// TwinCAT 3 PLC project PLC1
// ProgramVersion: 3.1.4026.19
// libraries:
//   Tc2_MC2, * (Beckhoff Automation GmbH)
//   Tc2_Standard, * (Beckhoff Automation GmbH)
//   Tc2_System, * (Beckhoff Automation GmbH)
// project tree:
//   GVLs/ Analog_Variables.TcGVL, Global_Variables.TcGVL, GVL_Axes.TcGVL
//   / PlcTask.TcTTO
//   POUs/ Analog_PRG.TcPOU, MAIN.TcPOU, Servo_Details.TcPOU, Step_3_Unscrambler.TcPOU, Step_4_EvenEnder.TcPOU, Step_5_Grading.TcPOU, Step_6_Log_Sequence.TcPOU, Step_7_Saw_Positioning.TcPOU, Step_8_Outfeed.TcPOU, Tower_Light_Manager.TcPOU, Step_1_TiltHoist.TcPOU, Step_2_StickMachine.TcPOU
// real-time tasks:
//   TASK PlcTask: cycle T#10ms, priority 20, ADS port 350
// motion (NC):
//   TASK NC-Task 1 SAF: cycle T#2ms, priority 4, ADS port 501
//   TASK NC-Task 1 SVB: cycle T#10ms, priority 8, ADS port 511
//   AXIS Axis 1 (id 1)
//     Dynamic: Acceleration=4141.08, Deceleration=4141.08, Jerk=45551.9
//     Velo: RefSearch=37.6461354666667, RefSync=37.6461354666667, SlowManual=188.230677333333, FastManual=1129.384064, Fast=3764.61354666667, Maximum=3764.61
//     PositionAreaControl: Enable=false
//     TargetPosControl: Range=0.5, Time=0.01
//     OtherSettings: AllowMotionCmdToSlave=true
//     encoder EncType=8
//       EncPara: ScaleFactorNumerator=104.8576, ScaleFactorDenominator=1048576, MaxCount=#xffffffff
//     drive DrvType=9
//       DrvPara: MaxCount=#xffffffff, DriveControlDWord=#x00030000
//         Analog: VeloReferenz=4141.07490133333, VeloScale=1.02398817080127, TorqueSetpointScale=10, ScaleFactorActTorque=0.1
//         TimeComp: TaskDelayCycles=1
//     controller CtrType=1
//       CtrPara: PriorControlFactor=1
//         PosDiffControl: Enable=false
//         PID: PosKp=10
//         Observer: BandWidth=20
// I/O:
//   DEVICE Device 1 (EtherCAT), AmsNetId 5.164.185.153.2.1
//     Term 1 (EK1100) [EK1100 EtherCAT Coupler (2A E-Bus)]
//       Term 2 (EL1417) [EL1417 32Ch. Dig. Input 24V]
//       Term 3 (EL2407) [EL2407 32Ch. Dig. Output 24V, 0.5A]
//       Term 9 (EL9011) [EL9011 End Terminal]
//     Drive 4 (AX5203-0000-0011) [AX5203-0000-0011 EtherCAT Drive (SoE, 2 Ch.)]
// variable links:
//   NC-Task 1 SAF/Axes/Axis 1 <-> Device 1 (EtherCAT)/Drive 4 (AX5203-0000-0011)
//     Drive/Inputs/In/nDcOutputTime <-> InfoData/DcOutputShift
//     Drive/Inputs/In/nState1 <-> AT 1/Drive status word @bit 8
//     Drive/Inputs/In/nState2 <-> AT 1/Drive status word
//     Drive/Inputs/In/nState4 @bit 1 <-> WcState/InputToggle
//     Drive/Inputs/In/nState4 <-> WcState/WcState
//     Drive/Outputs/Out/nCtrl1 <-> MDT 1/Master control word @bit 8
//     Drive/Outputs/Out/nDataOut2 <-> MDT 1/Velocity command value
//     Enc/Inputs/In/nDataIn1 <-> AT 1/Position feedback 1 value
//     Enc/Inputs/In/nDcInputTime <-> InfoData/DcInputShift
//     Enc/Inputs/In/nState4 @bit 1 <-> WcState/InputToggle
//     Enc/Inputs/In/nState4 <-> WcState/WcState
//   PLC1/PLC1 Instance <-> NC-Task 1 SAF/Axes/Axis 1
//     PlcTask Inputs/GVL_Axes.Axis1.NcToPlc <-> Outputs/ToPlc
//     PlcTask Outputs/GVL_Axes.Axis1.PlcToNc <-> Inputs/FromPlc

CONFIGURATION PLC1
    RESOURCE PLC ON TwinCAT3
        TASK PlcTask(INTERVAL := T#10ms, PRIORITY := 20);
        PROGRAM MAIN WITH PlcTask : MAIN;
        PROGRAM Step_1_TiltHoist WITH PlcTask : Step_1_TiltHoist;
        PROGRAM Step_2_StickMachine WITH PlcTask : Step_2_StickMachine;
        PROGRAM Step_3_Unscrambler WITH PlcTask : Step_3_Unscrambler;
        PROGRAM Step_4_EvenEnder WITH PlcTask : Step_4_EvenEnder;
        PROGRAM Servo_Details WITH PlcTask : Servo_Details;
        PROGRAM Step_5_Grading WITH PlcTask : Step_5_Grading;
        PROGRAM Step_6_Log_Sequence WITH PlcTask : Step_6_Log_Sequence;
        PROGRAM Step_7_Saw_Positioning WITH PlcTask : Step_7_Saw_Positioning;
        PROGRAM Step_8_Outfeed WITH PlcTask : Step_8_Outfeed;
    END_RESOURCE
END_CONFIGURATION

// ---- GVLs/Analog_Variables.TcGVL
VAR_GLOBAL
	

	AI_INT  : INT;   // from EL3255, 0.0–10.0 V
    AO_INT : INT;   // to EL4004, 0.0–10.0 V



















END_VAR

// ---- GVLs/Global_Variables.TcGVL
VAR_GLOBAL 
//--------------------------------- Power_Panel_IO---------------------------------


	//INPUTS for EL1409 (16 inputs avilable)
	SawPhotoeye AT %I*:BOOL;
	OutfeedRopePull AT %I*:BOOL;
	//Manual Motor Protector Signals//
	TiltHoistMMP AT %I*:BOOL;
	StickConveyorMMP AT %I*:BOOL; 
	StickFeedChainMMP AT %I*:BOOL; 
	EvenEnderMMP AT %I*:BOOL; 
	ScrapConveyorMMP AT %I*:BOOL; 
	OutFeedConveyorMMP AT %I*:BOOL;
	DustCollectorMMP AT %I*:BOOL;
	SawBlade1MMP AT %I*:BOOL;
	SawBlade2MMP AT %I*:BOOL;
	//Safety Singal
	SafetyCircuitSignal AT %I*:BOOL;
	
		//Servo
		OverTRavelLimitREV AT %I*:BOOL; 
		OverTRavelLimitFWD AT %I*:BOOL;
		HomingSensor AT %I*:BOOL;
	

	//INPUTS for EL1859 (8 inputs avilable)
	VFD1Faulted AT %I*:BOOL; //Unscrambler Chain
	VFD2Faulted AT %I*:BOOL; //Grading Chain 
	VFD3Faulted AT %I*:BOOL; //Feed Chain - Saw
	GradingEndLimit AT %I*:BOOL; // Grading end limit switch
	SawFeedChainHomingSensor AT %I*:BOOL; // saw feed chain homing sensor	
	
	//OUTPUTS for EL2409 (16 outputs avilable)
	ResetVFDs AT %Q*:BOOL;
	UnscramblerVFD1FWD AT %Q*:BOOL; //Unscrambler Chain FWD
	UnscramblerVFD1REV AT %Q*:BOOL; //Unscrambler Chain REV
	GradingVFD2FWD AT %Q*:BOOL; //Grading Chain 
	SawFeedChainVFD3FWD AT %Q*:BOOL; //Feed Chain - Saw
	
	TiltHoistFWD AT %Q*:BOOL;
	TiltHoistREV AT %Q*:BOOL;
	StickConveyorFWD AT %Q*:BOOL;
	StickFeedChainFWD AT %Q*:BOOL;
	EvenEnderFWD AT %Q*:BOOL;
	ScrapConveyorFWD AT %Q*:BOOL;
	OutFeedConveyorFWD AT %Q*:BOOL;
	DustCollectorFWD AT %Q*:BOOL;
	SawBladesFWD AT %Q*:BOOL;
	
	//OUTPUTS for EL1859 (8 outputs available)
	GradingVFD2REV AT %Q*:BOOL; //Grading Chain REV
	SawFeedChainVFD3REV AT %Q*:BOOL; //Feed Chain - Saw
	
	
	
//---------------------------------Control_Panel_IO----------------------------------

	
	//INPUTS for EL1409
	
	PBFoot:ARRAY[4..16] OF BOOL;
	
	ConfirmPB AT %I*:BOOL; //Confirms Board Input
	CancelPB AT %I*:BOOL; //Cancels Last Board Input
	//PanelStopPB AT %I*:BOOL; //CycleStopPB same input 
	
	//OUTPUTS for EL2409

	
	LTFoot:ARRAY[4..16]OF BOOL;

	
	//ANALOG INPUTS for EL3255
	AI_POT:INT;     // changed on the HMI screen
	
	//ANALOG OUTPUTS for EL4004
	UnscramblerVFD1speed:INT; //Unscrambler Chain
	GradingVFD2speed:INT; //Grading Chain 
	SawFeedVFD3speed:INT; //Feed Chain - Saw
		
	
	
	
	
//---------------------------------EtherCAT_Box_IO---------------------------------

	//INPUTS for EPP2339-0021
	TopLimitSwitch AT %I*:BOOL; //Tilt Hoist
	BottomLimitSwitch AT %I*:BOOL; //Tilt Hoist
	CycleStartPB AT %I*:BOOL; //Box for Tower Light
	CycleStopPB AT %I*:BOOL; //Box for Tower Light
	OpticalSensor AT %I*:BOOL; //Detects Board falling off Tilt Hoist
	StickMachine_TopLimit AT %I*:BOOL; //Top Limit Indicator for Stick Machine
	UnscramblerOpticalSensor AT %I*:BOOL; //Detects board at the bottom of Unscrambler/start of grading Line
	GradingRopePull AT %I*:BOOL; // Start/Stop Grading Chain Line 
	
	
	
	//OUTPUTS for EPP2339-0021
	RedLight AT %Q*:BOOL;
	YellowLight AT %Q*:BOOL;
	GreenLight AT %Q*:BOOL;
	StickMachine_Motor AT %Q*:BOOL; // Start/Stop motor for stick receiving machine, it wraps the sticks up on a sling or something
	
	
	
	
	
	
	//-------------------------------------------------INTERNALS----------------------------------------------------------------------------------------------------------
	
	
	//---------------------------------Tower Light Manager---------------------------------
	
	// Requests from steps (set in Step_1, Step_2, etc.)
    Step1_RedFlash  : BOOL;
    Step1_RedSteady : BOOL;
    Step2_RedFlash  : BOOL;
    Step2_RedSteady : BOOL;
	Step3_RedFlash  : BOOL;
    Step3_RedSteady : BOOL;
	Step5_RedFlash  : BOOL;
    Step5_RedSteady : BOOL;
	Step6_RedFlash  : BOOL;
    Step6_RedSteady : BOOL;
	Step7_RedFlash  : BOOL;
    Step7_RedSteady : BOOL;
	
	
    Step1_YellowSteady : BOOL;
	Step1_YellowFlash  : BOOL;
    Step2_YellowSteady : BOOL;
	Step2_YellowFlash  : BOOL;
	Step3_YellowSteady : BOOL;
	Step3_YellowFlash  : BOOL;
	Step5_YellowSteady : BOOL;
	Step5_YellowFlash  : BOOL;
	Step6_YellowSteady : BOOL;
	Step6_YellowFlash  : BOOL;
	Step7_YellowSteady : BOOL;
	Step7_YellowFlash  : BOOL;

 	Step1_GreenSteady : BOOL;
	Step1_GreenFlash  : BOOL;
    Step2_GreenSteady : BOOL;
	Step2_GreenFlash  : BOOL;
	Step3_GreenSteady : BOOL;
	Step3_GreenFlash  : BOOL;
	Step5_GreenSteady : BOOL;
	Step5_GreenFlash  : BOOL;
	Step6_GreenSteady : BOOL;
	Step6_GreenFlash  : BOOL;
	Step7_GreenSteady : BOOL;
	Step7_GreenFlash  : BOOL;	
	
	
	
	
	//--------------------------Auto/Manual Mode-------------------------------

	
	AutoMode : BOOL;	
	
	
	//--------------------------Permissives-------------------------------------
	
	
	Permissive : BOOL;
	
	
	//---------------------------States---------------------------------------
	
	GlobalState : INT :=0; 
	Step1_State : INT :=0;
	Step2_State : INT :=0;
	Step3_State : INT :=0;
	Step4_State : INT :=0;
	Step5_State : INT :=0;
	Step6_State : INT :=0;
	Step7_State : INT :=0;
	Step8_State : INT :=0;
	
	//---------------------------------Unscrambler------------------------------
	
	
	UnscramblerBoardDetected : BOOL;
	
	

	//------------------------------Timers------------------------------------
	
	
	
	UnscramblerDelay : TON;
	
	
	
	//--------------------------------misc----------------------------------
	
	
	Step2OffSignal : BOOL;
	StopStep3: BOOL;
	
	//--------------------------------Faults & Displays----------------------------------------
	
	
	Fault : ARRAY[1..10] OF BOOL;             // Faults and Displays are described in Main POU
	FaultDisplay : ARRAY[1..10] OF STRING[100];
	
	
	
	
	
	//-----------------------------------------Log Sequence------------------------------------

	ConfirmedFoot  : INT := 0;   // Confirmed length	
	FootFIFO : ARRAY[1..5] OF INT := [0, 0, 0, 0, 0];
	
	
	
	
	
	//---------------------------------Servo------------------------
	
	ServoInPosition : BOOL;
	HMI_GoToPosition : BOOL;
	
	
	
	
	//------------------------------Motion---------------------------------------------------
	//MC_Power
	fbMC_Power1: MC_Power;
	xEnable: BOOL;
	xControlPower: BOOL; //simulate control power
	fbMC_Power2: MC_Power;
	lrAxis2_Override: LREAL;
	
	//MC_Reset
	fbMC_Reset1: MC_Reset;
	xAxisReset: BOOL;
	fbMC_Reset2: MC_Reset;
	xMachineReset: BOOL;
	
	//Move_Relative
	fbMC_MoveRelative1: MC_MoveRelative;
	xExecuteDistanceRel: BOOL;
	lrDistance: LREAL := 10.0;
	
	//Move_Absolute
	fbMove_Absolute1: MC_MoveAbsolute;
	xExecuteDistanceAbs1: BOOL;
	lrTargetPosition: LREAL; //target posiiton
	fbMC_MoveVelocity1: MC_MoveVelocity;
	
	//Move_Velocity
	xExecuteMoveVelocity1: BOOL;
	
	//MC_Stop
	fbMC_Stop1: MC_Stop;
	xExecuteStop1: BOOL;
	
	//MC_Halt
	fbMC_Halt: MC_Halt;
	xExecuteHalt1: BOOL;
	fbMC_MoveJog1: MC_Jog;
	
	//MC_Home
	fbMC_Home1: MC_Home;
	xExecuteHome1: BOOL;
	xJogForward: BOOL;
	xJogBackwards: BOOL;
	
	
	//Other
	xMoveAbsDone1: BOOL;
	xMoveAbsBusy1: BOOL;
	lrActualPosition: LREAL;
	PositionTolerance       : LREAL := 0.05; // acceptable error window
	
	
END_VAR

// ---- GVLs/GVL_Axes.TcGVL
{attribute 'qualified_only'}
VAR_GLOBAL
	Axis1 : AXIS_REF;
	Axis2 : AXIS_REF;
END_VAR

// ---- POUs/MAIN.TcPOU
PROGRAM MAIN
VAR
	// --------------------------Tower Light Manager-----------------------
	Any_RedFlash  : BOOL;
    Any_RedSteady : BOOL;
    Any_YellowSteady : BOOL;
	 Any_YellowFlash : BOOL;
    Any_GreenSteady  : BOOL;
	Any_GreenFlash  : BOOL;
	Main_RedFlash : BOOL;
	

    TL : Tower_Light_Manager;
	
	rtBoardStuckatUnscrambler: BOOL;
	
	i : INT;
	
	 SafetyFallingEdgeDetect   : F_TRIG; // detects high→low transition

END_VAR


//-------------------------------------Defaults--------------------------------


 //--------------------------Tower Light Manager-----------------------

Any_RedFlash  := Step1_RedFlash  OR Step2_RedFlash  OR Step3_RedFlash OR Step5_RedFlash OR Step6_RedFlash OR Step7_RedFlash OR Main_RedFlash;
Any_RedSteady := Step1_RedSteady OR Step2_RedSteady OR Step3_RedSteady OR Step5_RedSteady OR Step6_RedSteady OR Step7_RedSteady;
Any_YellowSteady := Step1_YellowSteady OR Step2_YellowSteady OR Step3_YellowSteady OR Step5_YellowSteady OR Step6_YellowSteady OR Step7_YellowSteady;
Any_YellowFlash := Step1_YellowFlash OR Step2_YellowFlash OR Step3_YellowFlash OR Step5_YellowFlash OR Step6_YellowFlash OR Step7_YellowFlash;
Any_GreenSteady := Step1_GreenSteady OR Step2_GreenSteady OR Step3_GreenSteady OR Step5_GreenSteady OR Step6_GreenSteady OR Step7_GreenSteady;
Any_GreenFlash := Step1_GreenFlash OR Step2_GreenFlash OR Step3_GreenFlash OR Step5_GreenFlash OR Step6_GreenFlash OR Step7_GreenFlash;


// Call manager once per scan
TL(
    RedFlash    := Any_RedFlash,
    RedSteady   := Any_RedSteady,
    YellowSteady  := Any_YellowSteady,
	YellowFlash  := Any_YellowFlash,
    GreenSteady  := Any_GreenSteady,
	GreenFlash  := Any_GreenFlash,
    BlinkPeriod := T#500MS,
    RedOut      => RedLight,        //RedLight/YellowLight/GreenLight
    YellowOut   => YellowLight,     // to the real %Q outputs
    GreenOut    => GreenLight
);




//--------------------------------Permissive-----------------------------------


Permissive := SafetyCircuitSignal;

IF NOT Permissive THEN
	Main_RedFlash := TRUE;
ELSE
	Main_RedFlash := FALSE;
END_IF





rtBoardStuckatUnscrambler :=  UnscramblerDelay.Q;



//--------------------------------Faults & Displays--------------------------------------
Fault[1] := StickMachine_TopLimit;  // Stick machine bin full
Fault[2] := Main_RedFlash;   //Safety Circuit Open
(*Fault[3] := 
Fault[4] := 
Fault[5] := 
Fault[6] := 
Fault[7] := 
Fault[8] := 
Fault[9] := 
Fault[10] := *)


IF Fault[1] THEN
	FaultDisplay[1] :='StickMachine Full';
ELSE
	FaultDisplay[1] :='';	
END_IF

IF Fault[2] THEN
	FaultDisplay[2] :='Safety Circuit Open';
ELSE
	FaultDisplay[2] :='';	
END_IF




//------------------------------Fault Reset--------------------------

END_PROGRAM

// ---- POUs/Tower_Light_Manager.TcPOU
FUNCTION_BLOCK PUBLIC Tower_Light_Manager
VAR_INPUT
// Any steps that ask for the inputs below
	RedFlash  : BOOL;    
	RedSteady  : BOOL;  
    YellowSteady   : BOOL;
	YellowFlash  : BOOL;   
    GreenSteady     : BOOL; 
	GreenFlash    : BOOL;  
    BlinkPeriod  : TIME := T#500MS; // configurable
END_VAR
VAR_OUTPUT
	RedOut    : BOOL;
    YellowOut : BOOL;
    GreenOut  : BOOL;
END_VAR
VAR
	tBlink : TON;
    blink  : BOOL;
END_VAR

RedOut    := FALSE;
YellowOut := FALSE;
GreenOut  := FALSE;




//  only run while flashing
IF RedFlash OR YellowFlash OR GreenFlash THEN
	tBlink(IN := TRUE, PT := BlinkPeriod);
	IF tBlink.Q THEN
	blink := NOT blink;
	tBlink(IN := FALSE); // retrigger
	END_IF;
ELSE
	tBlink(IN := FALSE);   // stop timer when not flashing
	blink := FALSE;        
END_IF;





IF RedFlash THEN
    RedOut := blink;                   // flashing red
ELSIF RedSteady THEN
    RedOut := TRUE;                    // steady red
ELSIF YellowSteady THEN
    YellowOut := TRUE;                 // steady yellow
ELSIF YellowFlash THEN
    YellowOut := blink;                // flashing yellow
ELSIF GreenSteady THEN
    GreenOut := TRUE;                  // steady green
ELSIF GreenFlash THEN
    GreenOut := blink;                 // flashing green
ELSE
   YellowOut := TRUE;  // nothing requested -> YellowOut Default
END_IF;

END_FUNCTION_BLOCK

// ---- POUs/Step_1_TiltHoist.TcPOU
PROGRAM Step_1_TiltHoist // Tilt Hoist
VAR
    // Edge detectors
    rtStart : R_TRIG;      // Rising edge Cycle Start
    rtStop  : R_TRIG;      // Rising edge Cycle Stop
    ftPhotoEye    : F_TRIG;      // Falling edge on optical sensor

    // Timers 
    tPause  : TON;         // 10 second pause after each falling edge
	tStep2OFFSignal : TON;      // 
   
    

    // Internals 
    LocalSafety_1 : BOOL;         //  Local Safety Conditions   
	JOGTiltHoistFWD : BOOL;    // set from HMI
	JOGTiltHoistREV : BOOL;    // set from HMI
   
END_VAR

// Safety
LocalSafety_1 := TiltHoistMMP;

 
// Defaults: make outputs known each scan
Step1_RedFlash    := FALSE;
Step1_RedSteady    := FALSE;
Step1_YellowSteady := FALSE;
Step1_YellowFlash := FALSE;
Step1_GreenSteady  := FALSE;
Step1_GreenFlash  := FALSE;
TiltHoistFWD := FALSE;
TiltHoistREV := FALSE;

// Edge detect PBs and Optical falling edge
rtStart(CLK := CycleStartPB);
rtStop(CLK := CycleStopPB);
ftPhotoEye(CLK := OpticalSensor); // TRUE for one scan when optical goes 1 -> 0 (falling)


// Stop button or lost permissive or lost local safety → go to IDLE immediately
IF rtStop.Q OR NOT Permissive OR NOT LocalSafety_1 THEN
    Step1_State := 0; // IDLE
END_IF	

// unscramblerboard detected for a few seconds, turn off tilt hoist feeding it.
IF UnscramblerBoardDetected THEN
    Step1_State := 5; // Stop
END_IF	
	

// Stick machine top limit or step2 yellow flash, wait for operator, stickmachine is full		
IF StickMachine_TopLimit OR Step2_YellowFlash THEN
	Step1_State := 40;	
END_IF

// -------------------- Manual override (when AutoMode = FALSE) ------------------
IF NOT AutoMode THEN
    // Simple, safe manual jogs
    IF JOGTiltHoistFWD AND NOT JOGTiltHoistREV AND NOT TopLimitSwitch THEN
        TiltHoistFWD := TRUE;
    END_IF

    IF JOGTiltHoistREV AND NOT JOGTiltHoistFWD AND NOT BottomLimitSwitch THEN
        TiltHoistREV := TRUE;
    END_IF

    // Tower lights in manual: Yellow
    IF NOT AutoMode THEN
        Step1_YellowSteady := TRUE;
    END_IF

    RETURN;    // skips Auto sequence when in manual
END_IF

// -------------------- AUTO SEQUENCE --------------------
CASE Step1_State OF
    0:  // IDLE / READY / STOPPED
       
 		Step1_YellowSteady := TRUE; // IDLE / READY / STOPPED
		
		TiltHoistFWD := FALSE;
		TiltHoistREV := FALSE;
		
		// Make sure pause timer is reset while idle
        tPause(IN := FALSE);
		
			
        // Start cycle when forklift driver presses CycleStart
        IF rtStart.Q AND Permissive AND LocalSafety_1 THEN
            Step1_State := 10;  // begin Forward cycle
        END_IF
		
		
	5:  // STOPPED from step3 unscrambler board detected
       
 		Step1_GreenSteady := TRUE; // IDLE / READY / STOPPED
		
		TiltHoistFWD := FALSE;
		TiltHoistREV := FALSE;
		
		(*tStep2OffSignal(IN:= TRUE, PT := T#2M); // If board is detected for too long at the unscrambler then tilt hoist stops and timer start for stick machine to turn off
		Step2OffSignal := tStep2OffSignal.Q;	  // step2offsignal is global var and goes to step_2 case:10 conditions*)
			
        // Start cycle when forklift driver presses CycleStart
		
		IF NOT UnscramblerBoardDetected AND Permissive AND LocalSafety_1 THEN
            Step1_State := 10;  // begin Forward cycle
		END_IF
				
		

    10: // AUTO FWD (advance until optical falling edge, then pause)
	Step1_RedFlash    := FALSE;
	Step1_RedSteady    := FALSE;
	Step1_YellowSteady := FALSE;
	Step1_YellowFlash := FALSE;
	Step1_GreenSteady  := TRUE;
	Step1_GreenFlash  := FALSE;       // Running

        // Drive forward unless top limit TRUE
        IF NOT TopLimitSwitch THEN
            TiltHoistFWD := TRUE;
        END_IF

        // If the top is reached → go to return
        IF TopLimitSwitch THEN
            TiltHoistFWD := FALSE;
            Step1_State := 30; // reverse to bottom
			
        // Every falling edge of the optical sensor -> pause 10s, then continue
        ELSIF ftPhotoEye.Q THEN
            TiltHoistFWD := FALSE;
            Step1_State := 20; // pause state
        END_IF

    20: // PAUSE 10s after a layer drops
        Step1_GreenSteady := TRUE;
        tPause(IN := TRUE, PT := T#5S);

        IF tPause.Q THEN
            // Pause done -> continue forward again
            tPause(IN := FALSE);
            Step1_State := 10;
        END_IF

    30: // RETURN REVERSE to bottom at end of cycle
        Step1_GreenSteady := TRUE;

        IF NOT BottomLimitSwitch THEN
            TiltHoistREV := TRUE;
        ELSE
            TiltHoistREV := FALSE;
            Step1_State := 40; // reached bottom limit switch
        END_IF

    40: // COMPLETE: flash RED to signal done, wait for operator
        
    Step1_RedFlash    := FALSE;
	Step1_RedSteady    := FALSE;
	Step1_YellowSteady := FALSE;
	Step1_YellowFlash := TRUE;
	Step1_GreenSteady  := FALSE;
	Step1_GreenFlash  := FALSE;

        // Operator can press Start to begin a new auto cycle
        IF rtStart.Q AND Permissive AND LocalSafety_1 THEN
            Step1_YellowFlash := FALSE;
            Step1_State := 10;         // start next cycle forward
        END_IF

        
END_CASE

END_PROGRAM

// ---- POUs/Step_2_StickMachine.TcPOU
PROGRAM Step_2_StickMachine // Stick Machine
VAR
	
	// Internals 
	JOGStickConveyorFWD : BOOL;     // set from HMI
	JOGStickFeedChainFWD : BOOL;   // set from HMI
	LocalSafety_2: BOOL;             //Safety Conditions
	
	
	 // Edge detectors
    rtStart : R_TRIG;      // Rising edge Cycle Start
    rtStop  : R_TRIG;      // Rising edge Cycle Stop
	
	
	
	// Timers 
    tHoistPause  : TON;         // Running time for Stick conveyor and feed chain after tilt hoist reaches bottom limit switch
	
	
	
END_VAR

// Safety
LocalSafety_2 := StickConveyorMMP AND StickFeedChainMMP;



// Defaults: make outputs known each scan
Step2_RedFlash    := FALSE;
Step2_RedSteady    := FALSE;
Step2_YellowSteady := FALSE;
Step2_YellowFlash := FALSE;
Step2_GreenSteady  := FALSE;
Step2_GreenFlash  := FALSE;
StickConveyorFWD := FALSE;
StickFeedChainFWD := FALSE;


// Edge detect PBs and Optical falling edge
rtStart(CLK := CycleStartPB);
rtStop(CLK := CycleStopPB);


// Stop button or lost permissive or lost local safety → go to IDLE immediately
IF (rtStop.Q OR NOT Permissive OR NOT LocalSafety_2) THEN
    Step2_State := 0;        // IDLE
END_IF;




// -------------------- Manual override (when AutoMode = FALSE) ------------------
IF NOT AutoMode THEN
    // Simple, safe manual jogs
    IF JOGStickConveyorFWD  AND Permissive AND LocalSafety_2 THEN
        StickConveyorFWD := TRUE;
	ELSE
		StickConveyorFWD := FALSE;
    END_IF

    IF JOGStickFeedChainFWD AND Permissive AND LocalSafety_2 THEN
        StickFeedChainFWD := TRUE;
	ELSE
		StickFeedChainFWD := FALSE;
    END_IF

    // Tower lights in manual: Yellow
    IF NOT AutoMode THEN
        Step2_YellowSteady := TRUE;
    END_IF

    RETURN;    // skips Auto sequence when in manual
END_IF



    // ---------------------- Auto Sequence-------------------------------------

CASE Step2_State OF

    0:  // IDLE / READY
        Step2_YellowSteady := TRUE;
        StickConveyorFWD   := FALSE;
        StickFeedChainFWD  := FALSE;

        // If safe and not full, wait for Step 1 pause or start signal
        IF (Permissive AND LocalSafety_2 AND NOT StickMachine_TopLimit) THEN
            IF rtStart.Q THEN
                Step2_State := 10;      // start feeding
            END_IF
        END_IF


    // ---------------------------------------------------
    10: // RUNNING / FEEDING
     
		Step2_RedFlash    := FALSE;
		Step2_RedSteady    := FALSE;
		Step2_YellowSteady := FALSE;
		Step2_YellowFlash := FALSE;
		Step2_GreenSteady  := TRUE;
		Step2_GreenFlash  := FALSE;
        StickConveyorFWD  := TRUE;
        StickFeedChainFWD := TRUE;
		
		UnscramblerDelay(IN := UnscramblerBoardDetected, PT := T#30S);	
		 tHoistPause(IN := Step1_YellowFlash OR UnscramblerDelay.IN, PT := T#30S); // Tilt hoist reaches bottom limit and timer start, stickmachine motors run for set time after tilt hoist reaches bottom
		
        // Stop when bin becomes full or Tilt Hoist is at bottom
        IF StickMachine_TopLimit OR tHoistPause.Q (*OR Step2OffSignal*)THEN
            StickConveyorFWD  := FALSE;
            StickFeedChainFWD := FALSE;
			StopStep3 := TRUE;
            Step2_State := 20;          // go to FULL / FLASH
        END_IF

        // Lost safety or permissive → back to IDLE
        IF (NOT Permissive) OR (NOT LocalSafety_2) THEN
            StickConveyorFWD  := FALSE;
            StickFeedChainFWD := FALSE;
            Step2_State := 0;
        END_IF


    // ---------------------------------------------------
    20: // FULL BIN / Yellow FLASH
        Step2_RedFlash    := FALSE;
		Step2_RedSteady    := FALSE;
		Step2_YellowSteady := FALSE;
		Step2_YellowFlash := TRUE;
		Step2_GreenSteady  := FALSE;
		Step2_GreenFlash  := FALSE;
        StickConveyorFWD   := FALSE;
        StickFeedChainFWD  := FALSE;
		
       
        IF rtStart.Q AND NOT StickMachine_TopLimit AND Permissive AND LocalSafety_2 THEN
			Step2_YellowFlash := FALSE;
            Step2_State := 10;          // go to running
        END_IF


END_CASE

END_PROGRAM

// ---- POUs/Step_3_Unscrambler.TcPOU
PROGRAM Step_3_Unscrambler // Unscrambler
VAR
	//--------------------Internals--------------------
		LocalSafety_3  : BOOL;
    	tBoardDetect_3   : TON;   // duration before unscrambler stops
		
	
	
	
	
	//----------------------Manual Mode---------------------------	
 		JOGUnscramblerVFD1FWD : BOOL; //HMI
		JOGUnscramblerVFD1REV : BOOL;
	
		// Edge detectors
   	 	rtTiltHoistOptical_3 : R_TRIG;      // Rising edge on tilt hoist optical sensor
   		

	
	// duration of idle tilt hoist to stop unscrambler	
	tHoistIdle_3: TON;  
	tStopStep3: TON;
	
	
END_VAR

// ---------- local safety ----------

LocalSafety_3 := NOT VFD1Faulted;



// ---------- defaults ----------
Step3_RedFlash     := FALSE;
Step3_RedSteady    := FALSE;
Step3_YellowSteady := FALSE;
Step3_YellowFlash  := FALSE;
Step3_GreenSteady  := FALSE;
Step3_GreenFlash   := FALSE;

UnscramblerVFD1FWD := FALSE;
UnscramblerVFD1REV := FALSE;


(*rtTiltHoistOptical_3(CLK := OpticalSensor); // Rising edge each time the hoist sensor triggers

tHoistIdle_3(IN := NOT rtTiltHoistOptical_3.Q, PT := T#1M);*)

// ---------- Safety ----------
IF NOT Permissive OR NOT LocalSafety_3 OR UnscramblerDelay.Q OR CycleStopPB THEN
    Step3_State := 0;
END_IF


// ---------- sensor timing: stop if held > ----------
tBoardDetect_3(IN := UnscramblerOpticalSensor, PT := T#3S);
UnscramblerBoardDetected := tBoardDetect_3.Q;

// ---------- sensor timing: stop if held > ----------
tStopStep3(IN := Step1_YellowFlash, PT := T#30S);
StopStep3 := tStopStep3.Q;


// ----------------------------------------- Manual ---------------------------------------------------------

IF NOT AutoMode THEN
   
    IF JOGUnscramblerVFD1FWD AND LocalSafety_3 AND Permissive THEN
        UnscramblerVFD1FWD := TRUE;
    ELSE
        UnscramblerVFD1FWD := FALSE;
    END_IF;
	
    IF JOGUnscramblerVFD1REV AND LocalSafety_3 AND Permissive THEN
       UnscramblerVFD1REV := TRUE;
	ELSE  
		UnscramblerVFD1REV := FALSE; 
    END_IF;

 
 RETURN;   // skip auto sequence
END_IF;






//--------------------------------------------Auto Sequence-----------------------------------------------------------------
CASE Step3_State OF
// ---------------- IDLE ----------------
    0:
	
UnscramblerVFD1FWD := FALSE;
		
IF Permissive AND LocalSafety_3 AND OpticalSensor THEN
   Step3_State := 10; 
END_IF




// ---------------- RUNNING ----------------
    10:

UnscramblerVFD1FWD := TRUE;

// board detected at grader set time → stop
IF UnscramblerBoardDetected OR StopStep3 THEN
   UnscramblerVFD1FWD := FALSE;
   Step3_State := 20;  // stopped due to board
END_IF
   



        
// ---------------- STOPPED DUE TO BOARD or IDLE ------------------------------
    20:
        
UnscramblerVFD1FWD  := FALSE;
       
IF NOT UnscramblerBoardDetected THEN
	Step3_State := 10;
END_IF
        
	

END_CASE

END_PROGRAM

// ---- POUs/Step_4_EvenEnder.TcPOU
PROGRAM Step_4_EvenEnder // Even Ender
VAR
	//-----------------Safety------------------
	LocalSafety_4 : BOOL;
	

END_VAR

// ---------- local safety ----------
LocalSafety_4 := EvenEnderMMP;

// ---------- defaults ----------

EvenEnderFWD := FALSE;


// ---------- Safety ----------
IF NOT Permissive OR NOT LocalSafety_4 THEN   // if anything unsafe, force the system to IDLE (state 0).
    Step4_State := 0;
END_IF



// -------------------------------Main sequence ---------------------------------
CASE Step4_State OF
// ---------------- IDLE/STOPPED ----------------
0: 
	
	EvenEnderFWD := FALSE;
	   
IF GradingVFD2FWD THEN         // Transition to RUN when the upstream grading conveyor (GradingVFD2) is running
	Step4_State := 10;
END_IF
	
	
	
// ----------------------- RUN ----------------------	
10:
	
	EvenEnderFWD := TRUE;     //EvenEnder motor to run forward.
	
IF NOT GradingVFD2FWD OR NOT Permissive OR NOT LocalSafety_4 THEN       // Return to IDLE if the upstream conveyor stops, or if a permissive/localsafety input is lost.
	EvenEnderFWD := FALSE;	
	Step4_State := 0;
		
END_IF
	
	
	
	
	
	
	
	
	
	
	
	
	
	
	
	
	
	
	
END_CASE

END_PROGRAM

// ---- POUs/Servo_Details.TcPOU
PROGRAM Servo_Details
VAR
	
END_VAR

// -----------------------------------Motion--------------------------------------
//Read Status
	GVL_Axes.Axis1.ReadStatus();


//Enable
	IF xControlPower THEN
		xEnable := TRUE;
	ELSE
		xEnable := FALSE;	
	END_IF

fbMC_Power1(
		Axis:= GVL_Axes.Axis1, 
		Enable:= xEnable, // Typically controlled by the machine control power or something similar
		Enable_Positive:= xEnable, // should be tied to front and back limit switches, if limit true then one direction should be false.-------------------------------------------MODIFY-----------------------
		Enable_Negative:= xEnable, 
		Override:= 100);  //It’s like a “speed knob” that adjusts all moves without rewriting motion commands. Feedrate override — scales all commanded velocities by this percentage.Type: LREAL (real number, typically 0–100%)


(*		BufferMode:= , Determines how new motion commands are handled when another one is already active.
		Options:= , 
		Status=> , Reports that the axis is successfully enabled.
		Busy=> , Indicates the function block is currently executing the command.
		Error=> , Goes TRUE when the function block or NC reports an error.
		ErrorID=> ); Numerical error code providing details about what failed.Always log ErrorID when troubleshooting — it’s your direct clue.
*)



//Reset

IF xMachineReset THEN
	xAxisReset := TRUE;
ELSE
	xAxisReset := FALSE;
END_IF




fbMC_Reset1(
	Axis:= GVL_Axes.Axis1, 
	Execute:= xAxisReset AND GVL_Axes.Axis1.Status.Error); // command will not be issued unless there is an error
	

(*	
	Done=> , //TRUE for one cycle when reset completes
	Busy=> , //TRUE while reset is running
	Error=> , //TRUE if reset fails
	ErrorID=> ); //Motion library error code		
*)		
	
	
//Move_Relative


fbMC_MoveRelative1(
		Axis:= GVL_Axes.Axis1, 
		Execute:= xExecuteDistanceRel, // Rising edge (FALSE → TRUE) starts the relative move. Keep it TRUE while you want the command to remain active; drop it to FALSE after Done or Error if you’re pulsing it.
		Distance:= lrDistance, //Units are whatever your axis units are (e.g. mm, degrees, revs). Positive = forward, negative = reverse. Target = ActPos + Distance.
		Velocity:= 5.0); //Peak speed of your move. Needs to be within axis limits; too high can cause faults or be clamped.
(*
		Acceleration:= , //How fast it ramps up to Velocity. Too high → potential following error / torque limits. Too low → sluggish motion.
		Deceleration:= , //How fast it slows down from Velocity to 0. Similar considerations as Accel.
		Jerk:= , //Optional. If supported, higher jerk = sharper ramps; lower jerk = smoother, more gentle motion. Often set to 0 or a default at first.
		BufferMode:= , //mcAborting (default: stop current then do this), mcBuffered (queue after current), mcBlendingLow / mcBlendingPrevious (smooth transitions). For simple testing, stick with mcAborting.
		Options:= , 
		Done=> , //TRUE when the move has reached its target and the command is complete. Typically goes TRUE for at least one cycle.
		Busy=> , //TRUE from the moment the move starts until it’s finished or aborted. If Busy = TRUE, the command is still active.
		Active=> , //TRUE while this specific move is the one controlling the axis. Useful if you chain/buffer multiple moves.
		CommandAborted=> , //TRUE if the move got cancelled by another command (Stop, new move with mcAborting, etc.). Not an error — just means “I was told to stop early.”
		Error=> , //TRUE if something went wrong (limit reached, following error, accel/velocity too high, drive fault, etc.).
		ErrorID=> ); //Tells you what error occurred. Log or show this in HMI; use docs to decode (e.g. following error, limit exceeded, axis not enabled, etc.).
*)




//Move_Absolute

fbMove_Absolute1(
		Axis:= GVL_Axes.Axis1, 
		Execute:= xExecuteDistanceAbs1, 
		Position:= lrTargetPosition, 
		Velocity:= 1.0, 
		Acceleration:= , 
		Deceleration:= , 
		Jerk:= , 
		BufferMode:= , 
		Options:= , 
		Done=> xMoveAbsDone1, 
		Busy=> xMoveAbsBusy1, 
		Active=> , 
		CommandAborted=> , 
		Error=> , 
		ErrorID=> );		
		
	
		
//Move_Velocity

fbMC_MoveVelocity1(
		Axis:= GVL_Axes.Axis1 , 
		Execute:= xExecuteMoveVelocity1, 
		Velocity:= 250, 
		Acceleration:= , 
		Deceleration:= , 
		Jerk:= , 
		Direction:= , 
		BufferMode:= , 
		Options:= , 
		InVelocity=> , 
		Busy=> , 
		Active=> , 
		CommandAborted=> , 
		Error=> , 
		ErrorID=> );
		
//MC_Halt 

fbMC_Halt(
	Axis:= GVL_Axes.Axis1, //MC_Halt = “panic brake, then let go.” Even if held TRUE, move executions can still go TRUE.
	Execute:= xExecuteHalt1, 
	Deceleration:= , 
	Jerk:= , 
	BufferMode:= , 
	Options:= , 
	Done=> , 
	Busy=> , 
	Active=> , 
	CommandAborted=> , 
	Error=> , 
	ErrorID=> );
//MC_Stop

fbMC_Stop1( //Typically used for E-Stop
	Axis:= GVL_Axes.Axis1, //If MC_Stop.Execute stays TRUE, it keeps the axis locked
	Execute:= xExecuteStop1,
	Deceleration:= , 
	Jerk:= , 
	Options:= , 
	Done=> , 
	Busy=> , 
	Active=> , 
	CommandAborted=> , 
	Error=> , 
	ErrorID=> );
	

//MC_Jog

fbMC_MoveJog1(
	Axis:= GVL_Axes.Axis1, 
	JogForward:= xJogForward, 
	JogBackwards:= xJogBackwards, 
	Mode:= E_JogMode.MC_JOGMODE_STANDARD_SLOW, 
	Position:= , 
	Velocity:= , 
	Acceleration:= , 
	Deceleration:= , 
	Jerk:= , 
	Done=> , 
	Busy=> , 
	Active=> , 
	CommandAborted=> , 
	Error=> , 
	ErrorID=> );
	

//MC_Home

fbMC_Home1(
	Axis:= GVL_Axes.Axis1, 
	Execute:= xExecuteHome1, 
	Position:= DEFAULT_HOME_POSITION, 
	HomingMode:= MC_Direct, 
	BufferMode:= , 
	Options:= , 
	bCalibrationCam:= , 
	Done=> , 
	Busy=> , 
	Active=> , 
	CommandAborted=> , 
	Error=> , 
	ErrorID=> );

END_PROGRAM

// ---- POUs/Step_5_Grading.TcPOU
PROGRAM Step_5_Grading //Grading Line
VAR
//--------------------Internals--------------------
	LocalSafety_5  : BOOL;
	
	
	
	
//----------------------Manual Mode---------------------------	
 		JOGGradingVFD2FWD : BOOL; //HMI
		JOGGradingVFD2REV : BOOL;	
	
	
	
// Edge detectors
    rtPullRope_5 : R_TRIG;      // Rising edge Pull Rope	
	
	
	
	
	
	
	
	
	
	
	
	
	
	
	
	
	
	
	
	
END_VAR

//----------------------Safety--------------------

LocalSafety_5  := NOT VFD2Faulted;


//---------------------Defaults-------------------

Step5_RedFlash    := FALSE;
Step5_RedSteady    := FALSE;
Step5_YellowSteady := FALSE;
Step5_YellowFlash := FALSE;
Step5_GreenSteady  := FALSE;
Step5_GreenFlash  := FALSE;
GradingVFD2FWD := FALSE;
GradingVFD2REV := FALSE;

rtPullRope_5(CLK := GradingRopePull);


// Stop button or lost permissive or lost local safety → go to IDLE immediately
IF CycleStopPB OR NOT Permissive OR NOT LocalSafety_5 THEN
    Step5_State := 0; // IDLE
END_IF	



// ----------------------------------- Manual override (when AutoMode = FALSE) ---------------------------------------
IF NOT AutoMode THEN
    GradingVFD2FWD := FALSE;
    GradingVFD2REV := FALSE;

    IF Permissive AND LocalSafety_5 THEN
        // Only run FWD if REV jog is NOT pressed
        IF JOGGradingVFD2FWD AND NOT JOGGradingVFD2REV THEN
            GradingVFD2FWD := TRUE;
        END_IF

        // Only run REV if FWD jog is NOT pressed
        IF JOGGradingVFD2REV AND NOT JOGGradingVFD2FWD THEN
            GradingVFD2REV := TRUE;
        END_IF
    END_IF;

    RETURN;
END_IF



//--------------------------AutoMode---------------------------------------------------------------------------
CASE Step5_State OF

0: // Stopped  


GradingVFD2FWD := FALSE;
GradingVFD2REV := FALSE;

IF CycleStartPB OR rtPullRope_5.Q THEN
    Step5_State := 5; // IDLE
END_IF	


5: // Running/Standby
   

IF NOT GradingEndLimit THEN
   GradingVFD2FWD := TRUE;   // start running
ELSE
	GradingVFD2FWD := FALSE;
END_IF;


IF rtPullRope_5.Q THEN
	Step5_State := 0;

END_IF





END_CASE;

END_PROGRAM

// ---- POUs/Step_6_Log_Sequence.TcPOU
PROGRAM Step_6_Log_Sequence
VAR
	j, i: INT;
	
	SelectedFoot   : INT := 0;   // 0 = none, otherwise 4..16
    //GVL ---------ConfirmedFoot  : INT := 0;   // Confirmed length
    rtConfirm      : R_TRIG;     // for one-shot on ConfirmPB
	rtCancel : R_TRIG;   // edge detector for Cancel
END_VAR





// One-shot on Confirm button
rtConfirm(CLK := ConfirmPB);
// One-shot on Cancel button
rtCancel(CLK := CancelPB);







// If a PB is pressed, set that light ON and others OFF
FOR j := 4 TO 16 DO
    IF PBFoot[j] THEN
        // turn all lights off first
        FOR i := 4 TO 16 DO
            LTFoot[i] := FALSE;
        END_FOR;
		
        // turn only this one ON
        LTFoot[j] := TRUE;
		
		// remember which length is selected
        SelectedFoot := j;   // j will be 4..16
    END_IF;
END_FOR;

//-------------------------------------------------------------------------------------

// One-shot on Confirm button
IF rtConfirm.Q THEN
    // Save the current selected length
    ConfirmedFoot := SelectedFoot;

    // Add it into the FIFO (first empty slot)
    FOR i := 1 TO 5 DO
        IF FootFIFO[i] = 0 THEN
            FootFIFO[i] := ConfirmedFoot;   // store new graded length
            EXIT;                           // stop after writing one slot
        END_IF;
    END_FOR;

    // 3) Clear the lights and selection ready for next board
    FOR j := 4 TO 16 DO
        LTFoot[j] := FALSE;
    END_FOR;

    SelectedFoot := 0;
END_IF;
	
//-----------------------------------------------------------------------------------
// One-shot on Cancel button
IF rtCancel.Q THEN
    // Remove the newest board entered by the grader.
    //  start from the back (slot 5) and clear the first non-zero we find.
    FOR i := 5 TO 1 BY -1 DO
        IF FootFIFO[i] <> 0 THEN // <> "Not equal to"
            FootFIFO[i] := 0;          // clear that newest entry
            EXIT;                      // stop after clearing one
        END_IF;
    END_FOR;
END_IF;

END_PROGRAM

// ---- POUs/Step_7_Saw_Positioning.TcPOU
PROGRAM Step_7_Saw_Positioning
VAR
	 i : INT;
	NextTargetLength: INT :=0;
	ActiveLength: INT;
	
	
	ftCutDone: F_TRIG;
	ftGradingEndLimit: F_TRIG;
	rtSawFeedChainHomingSensor : R_TRIG;
	rtGoToPosition : R_TRIG;
	rtExecuteAbs1 : R_TRIG;
	
	
	

	
	LocalSafety_7: BOOL;
END_VAR

//------------------Defaults--------------------

SawFeedChainVFD3FWD := FALSE;


// ---------- Safety ----------

LocalSafety_7 := NOT VFD3Faulted AND SawBlade1MMP AND SawBlade2MMP AND DustCollectorMMP;



IF NOT Permissive OR NOT LocalSafety_7 OR CycleStopPB THEN
    Step7_State := 0;
END_IF

//------------------Triggers------------------------------
ftCutDone(CLK := SawPhotoeye); 
rtGoToPosition(CLK := HMI_GoToPosition);
rtExecuteAbs1(CLK := xExecuteDistanceAbs1);


lrActualPosition := GVL_Axes.Axis1.NcToPlc.ActPos;



IF ftCutDone.Q THEN
    FOR i := 1 TO 4 DO
        FootFIFO[i] := FootFIFO[i + 1];
    END_FOR;
    FootFIFO[5] := 0;
END_IF;




//----------------------------------------Board Transfer---------------------------------


// ---------- Trigger to enter POSITIONING (state 0) ----------
IF ftCutDone.Q OR rtGoToPosition.Q THEN // falling edge on SawPhotoeye or HMI button "go to position" 
    Step7_State := 5;
END_IF






// ---------- State machine ----------
CASE Step7_State OF
	
0: // standby


SawFeedChainVFD3FWD := FALSE;
SawBladesFWD := FALSE;
DustCollectorFWD := FALSE;


IF CycleStartPB THEN
	Step7_State := 5;
END_IF





5:  // POSITIONING DECISION

SawBladesFWD := TRUE;
DustCollectorFWD := TRUE;

lrTargetPosition := FootFIFO[1]; // target position from queue

// If there’s no target length, do nothing
IF FootFIFO[1] = 0 THEN
    SawFeedChainVFD3FWD := FALSE;	
ELSE                  
	// Otherwise, continue with positioning logic
	// call FB every scan (Execute FALSE by default here)
        fbMove_Absolute1(
            Axis         := GVL_Axes.Axis1,
            Execute      := FALSE,
            Position     := lrTargetPosition,
            Velocity     := 3500.0,
            Acceleration := ,
            Deceleration := ,
            Jerk         := ,
            BufferMode   := MC_BufferMode.MC_Aborting,
            Options      := ,
	);

	// 1) Check if already at position
	IF ABS(lrActualPosition - lrTargetPosition) <= PositionTolerance (*LREAL := 0.05; // acceptable error window*) THEN
	// already in position, skip move
     Step7_State := 10; // back to feeding
	ELSE
	// 2) Execute a move if not yet in position
    Step7_State := 15; // Execute absolute trget position
	END_IF;
								
END_IF

10: //busy //running// FEEDING 


xExecuteDistanceAbs1:= FALSE;  


// still call FB to keep status fresh
        fbMove_Absolute1(
            Axis         := GVL_Axes.Axis1,
            Execute      := FALSE,
            Position     := lrTargetPosition,
            Velocity     := 3500.0,
            Acceleration := ,
            Deceleration := ,
            Jerk         := ,
            BufferMode   := MC_BufferMode.MC_Aborting,
            Options      := ,
);


SawFeedChainVFD3FWD := TRUE;
 
  // The edges at top will kick us back to state 0
  // when SawPhotoeye falls or HMI_GoToPos is pressed.
 

 
 15: //ISSUE MOVE (one-scan pulse), then wait for done

 
SawFeedChainVFD3FWD := FALSE;     
xExecuteDistanceAbs1:= TRUE;   // pulse Execute
           
       

// Call the motion block
fbMove_Absolute1(
	Axis         := GVL_Axes.Axis1,
	Execute      := rtExecuteAbs1.Q,
	Position     := lrTargetPosition,
	Velocity     := 3500.0,
	Acceleration := ,
	Deceleration := ,
	Jerk         := ,
	BufferMode   := MC_BufferMode.MC_Aborting,
	Options      := ,
);

// When the move is finished...
IF xMoveAbsDone1 THEN
   Step7_State  := 10;  
END_IF;


       

END_CASE

END_PROGRAM

// ---- POUs/Step_8_Outfeed.TcPOU
PROGRAM Step_8_Outfeed
VAR
// ------------triggers-----------------	
rtPullRope_8 : R_TRIG;



//--------safety---------------------
LocalSafety_8: BOOL;
	
	
	
	
END_VAR



//----------------------Safety--------------------

LocalSafety_8 := OutFeedConveyorMMP;


//---------------------Defaults-------------------


rtPullRope_8(CLK := OutfeedRopePull);


// Stop button or lost permissive or lost local safety → go to IDLE immediately
IF CycleStopPB OR NOT Permissive THEN
    Step5_State := 0; // IDLE
END_IF	



// ----------------------------------- Manual override (when AutoMode = FALSE) ---------------------------------------
IF NOT AutoMode THEN
    OutFeedConveyorFWD := FALSE;
	
    IF Permissive AND LocalSafety_8 THEN
        // Only run FWD if REV jog is NOT pressed
        IF OutFeedConveyorFWD THEN
            GradingVFD2FWD := TRUE;
		ELSE
			OutFeedConveyorFWD := FALSE;
        END_IF

    END_IF;

    RETURN;
END_IF



//--------------------------AutoMode---------------------------------------------------------------------------
CASE Step8_State OF

0: // Stopped  


OutFeedConveyorFWD := FALSE;


IF CycleStartPB OR rtPullRope_8.Q THEN
    Step5_State := 5; // IDLE
END_IF	


5: // Running/Standby
   
OutFeedConveyorFWD := TRUE;

IF rtPullRope_8.Q THEN
	Step5_State := 0;

END_IF





END_CASE;

END_PROGRAM

// ---- POUs/Analog_PRG.TcPOU
PROGRAM Analog_PRG
VAR
	

AI_Input : INT;
AO_Output : INT;
AO_Unscrambler : INT;
AO_Grading : INT;
AO_SawFeedChain: INT;

// --- Analog routing logic ---
// Selection = 1..3 (from HMI dropdown)
Selection : ARRAY[1..3] OF BOOL;  // 1=Unscrambler, 2=Grading, 3=SawFeed



END_VAR

//---------------------------Defaults-----------------------------
AO_Unscrambler := 0;
AO_Grading := 0;
AO_SawFeedChain := 0;



AI_INT := AI_Input;

UnscramblerVFD1speed := AO_Unscrambler;
GradingVFD2speed := AO_Grading;
SawFeedVFD3speed := AO_SawFeedChain;







CASE Selection OF
//Selection 1 - Unscrambler	
1:  

AO_Unscrambler := AI_Input;
AO_Grading := 0;
AO_SawFeedChain := 0;

// Selection 2 - Grading
2:  

AO_Grading := AI_Input;
AO_Unscrambler := 0;
AO_SawFeedChain := 0;


// Selection 3 - Saw FeedChain
3:  

AO_SawFeedChain := AI_Input;
AO_Unscrambler := 0;
AO_Grading := 0;

// --- Default (nothing selected) ---
ELSE
    AO_Unscrambler := 0;
    AO_Grading := 0;
    AO_SawFeedChain := 0;

END_CASE

END_PROGRAM
